{attribute addProperty BoxType "EL5151-0000-0020"}
{attribute addProperty Id "StatusAT %I*Status_08B4C8AD1621Counter_valueAT %I*UINT16217Latch_valueAT %I*UINT16218"}
{attribute addProperty CRC "697647136"}
{attribute addProperty SizeInBites "48"}
{attribute addProperty SizeInBytes "6"}
TYPE ENC_Inputs_29954020 :
STRUCT
	{attribute addProperty Name "Status"}
	Status AT %I* : Status_08B4C8AD;
	{attribute addProperty Name "Counter_value"}
	Counter_value AT %I* : UINT;
	{attribute addProperty Name "Latch_value"}
	Latch_value AT %I* : UINT;
END_STRUCT
END_TYPE

(* stored: Version 1.2.0.0, ProductVersion 3.1.4024.9
   DUT ENC_Inputs_29954020: Id {fe407083-fe88-4e03-a355-38fafe419d51} *)
